(* PLC project Tc2_MC2.MC_MoveModulo Demo, tc3-libraries-kb TwinCAT 3.1 *)
(* stored: creationDateTime 2026-05-21T00:00:00, modificationDateTime 2026-05-21T00:00:00 *)

PROGRAM P_Demo_MC_MoveModulo
  VAR
    fbIndexRotate : MC_MoveModulo;
    axisIndexTable : AXIS_REF;
    rtNextStation : R_TRIG;
    bAdvanceStation : BOOL := FALSE;  (* 在线 TRUE 一次 = 转到下一工位 *)
    lrNextStationDeg : LREAL := 90.0;  (* 下一工位的模数目标角度 *)
    bRotateDone : BOOL;
    nErrorID : UDINT;
  END_VAR

// =============================================================================
// 场景：4 工位分度盘 — 每按一次"下一工位"按钮，转台正向转 90° 到下一工位。
// 价值：模数 FB 处理角度 wrap，业务不用算"现位 + 90 是否过 360"。
// 验证：登录后 bAdvanceStation := TRUE 一次 → 角度 0→90；再触发 90→180；
//       连续 4 次回到 0；将 lrNextStationDeg 改为 720 看到转 2 圈再到位。
// =============================================================================

rtNextStation(CLK := bAdvanceStation);

fbIndexRotate(
    Execute      := rtNextStation.Q,
    Position     := lrNextStationDeg,
    Velocity     := 180.0,
    Acceleration := 360.0,
    Deceleration := 360.0,
    Jerk         := 3600.0,
    Direction    := MC_Positive_Direction,
    BufferMode   := MC_Aborting,
    Axis         := axisIndexTable,
    Done         => bRotateDone,
    ErrorID      => nErrorID
);
END_PROGRAM
